{attribute 'Tc2GvlVarNames'}
{attribute 'strict'}
//Disposizione Fotocellula Di Presenza in WA
TYPE e_Disposizione_FTC_WA :
(
	NOT_DEFINED			:= -1,
	FTC_PRESENZA_ANGOLO_DX	 := 1,	(* Identifica che la fotocellula di presenza della WorkArea è disposta nell'angolo a DX della WorkArea stessa *)
	FTC_PRESENZA_CENTRALE	 := 2,	(* Identifica che la fotocellula di presenza della WorkArea è disposta sulla mediana della WorkArea stessa *)	
	FTC_PRESENZA_ANGOLO_SX	 := 3	(* Identifica che la fotocellula di presenza della WorkArea è disposta nell'angolo a SX della WorkArea stessa *)
);
END_TYPE
//  NOT_DEFINED = '-1'

(* stored: Version 1.1.0.1, ProductVersion 3.1.4024.11
   EnumerationTextList e_Disposizione_FTC_WA: Id {49f39eaa-f69a-407e-8595-f4e6aa9d84f0} *)
